(* IEC 61131-3 sources: Elmo_Master/Lasal_PRG/Elmo_EtherCAT_Test_4Axis/Class/GL_9086_1_Slot00, 1 file *)

(* ---- GL_9086_1_Slot00.st ---- *)
//{{ECAT_DEFINES
#define GL_9086_1_SLOT00_ETHERCATSLAVE_PRODUCT_CODE 1196692218
#define GL_9086_1_SLOT00_ETHERCATSLAVE_VENDOR_ID    669
#define GL_9086_1_SLOT00_INPUTS_BYTE0_INDEX		16#6000
#define GL_9086_1_SLOT00_INPUTS_BYTE0_SUBINDEX			1
#define GL_9086_1_SLOT00_INPUTS_BYTE1_INDEX		16#6000
#define GL_9086_1_SLOT00_INPUTS_BYTE1_SUBINDEX			2
#define GL_9086_1_SLOT00_INPUTS_BYTE2_INDEX		16#6000
#define GL_9086_1_SLOT00_INPUTS_BYTE2_SUBINDEX			3
#define GL_9086_1_SLOT00_INPUTS_BYTE3_INDEX		16#6000
#define GL_9086_1_SLOT00_INPUTS_BYTE3_SUBINDEX			4
//}}ECAT_DEFINES

(*!
<Class
	Name               = "GL_9086_1_Slot00"
	Revision           = "0.0"
	RealtimeTask       = "false"
	CyclicTask         = "false"
	BackgroundTask     = "false"
	Sigmatek           = "false"
	OSInterface        = "false"
	HighPriority       = "false"
	Automatic          = "false"
	UpdateMode         = "Prescan"
	SharedCommandTable = "true"
	Objectsize         = "(600,120)"
	Comment            = "GT-12FA">
	<Channels>
		<Server Name="InputS_Byte0" Visualized="false" Initialize="false" WriteProtected="true" Retentive="false" Comment="Input(s)"/>
		<Server Name="InputS_Byte1" Visualized="false" Initialize="false" WriteProtected="true" Retentive="false" Comment="Input(s)"/>
		<Server Name="InputS_Byte2" Visualized="false" Initialize="false" WriteProtected="true" Retentive="false" Comment="Input(s)"/>
		<Server Name="InputS_Byte3" Visualized="false" Initialize="false" WriteProtected="true" Retentive="false" Comment="Input(s)"/>
	</Channels>
	<Network Name="GL_9086_1_Slot00">
		<!-- List of Components in this network -->
		<Components>
			<Object
				Name       = "_base"
				Class      = "ECAT_SlotBase"
				Position   = "(218,120)"
				Visualized = "true"
				Remotely   = "true">
				<Channels>
					<Server Name="ClassState"/>
					<Client Name="ECATSlotIn"/>
					<Client Name="Required" Value="1"/>
					<Client Name="Slot"/>
					<Client Name="SlotIndexInc" Value="0"/>
					<Client Name="ToStdLib"/>
					<Client Name="UseSlotIndexInc" Value="0"/>
				</Channels>
				<AdditionalData>
					<Entry Name="DeviceType" Value="ECAT_SlotBase"/>
					<Entry Name="HWKey" Value="HWD:M_ETHERCAT_MODULE:1:1:0"/>
				</AdditionalData>
			</Object>
		</Components>
		<Comments>
		</Comments>
		<!-- List of Connections in this network -->
		<Connections>
			<Connection Source="this.ClassState" Destination="_base.ClassState" Vertices="(902,210),(730,210),"/>
			<Connection Source="_base.ECATSlotIn" Destination="this.ECATSlotIn" Vertices="(218,210),(38,210),"/>
			<Connection Source="_base.Slot" Destination="this.Slot" Vertices="(218,270),(38,270),"/>
			<Connection Source="_base.SlotIndexInc" Destination="this.SlotIndexInc" Vertices="(218,330),(38,330),"/>
			<Connection Source="_base.UseSlotIndexInc" Destination="this.UseSlotIndexInc" Vertices="(218,390),(38,390),"/>
		</Connections>
		<!-- Headerfiles -->
		<Options>
		</Options>
	</Network>
	<ECAT_SlotModule Type="GT-12FA" ModuleVendor="669" ModuleIdent="1196692218" FileName="..\Runtime\HWConfig\ESI\Crevis EtherCAT IO Module\Crevis_GT-xxxx_V14.xml"/>
	<ECAT_SlotInfoData Type="0" Index="0"/>
</Class>
*)
#pragma using ECAT_SlotBase

GL_9086_1_Slot00 : CLASS
: ECAT_SlotBase
  //Servers:
	InputS_Byte0 	: SvrCh_DINT;
	InputS_Byte1 	: SvrCh_DINT;
	InputS_Byte2 	: SvrCh_DINT;
	InputS_Byte3 	: SvrCh_DINT;
  //Clients:
  //Variables:
  //Functions:
				//! <Function Comment="Overwrite in derived class to set the pdo settings" Name="SetPDOSettings"/>
	FUNCTION VIRTUAL GLOBAL SetPDOSettings
		VAR_OUTPUT
			retcode 	: DINT;
		END_VAR;
  //Tables:
	FUNCTION @STD
		VAR_OUTPUT
			ret_code	: CONFSTATES;
		END_VAR;
	FUNCTION GLOBAL TAB @CT_;
END_CLASS;

FUNCTION VIRTUAL GLOBAL GL_9086_1_Slot00::SetPDOSettings
	VAR_OUTPUT
		retcode 	: DINT;
	END_VAR

	retcode := ECAT_SlotBase::SetPDOSettings();
	if retcode <> 0 then
		return;
	end_if;

	retcode := AddPDOEntry(ECAT_PDO_TYPE_INPUT, #InputS_Byte0.dData, GL_9086_1_SLOT00_INPUTS_BYTE0_INDEX, GL_9086_1_SLOT00_INPUTS_BYTE0_SUBINDEX);
	if retcode <> 0 then
		AddPDOEntryFailed(retcode);
		return;
	end_if;

	retcode := AddPDOEntry(ECAT_PDO_TYPE_INPUT, #InputS_Byte1.dData, GL_9086_1_SLOT00_INPUTS_BYTE1_INDEX, GL_9086_1_SLOT00_INPUTS_BYTE1_SUBINDEX);
	if retcode <> 0 then
		AddPDOEntryFailed(retcode);
		return;
	end_if;

	retcode := AddPDOEntry(ECAT_PDO_TYPE_INPUT, #InputS_Byte2.dData, GL_9086_1_SLOT00_INPUTS_BYTE2_INDEX, GL_9086_1_SLOT00_INPUTS_BYTE2_SUBINDEX);
	if retcode <> 0 then
		AddPDOEntryFailed(retcode);
		return;
	end_if;

	retcode := AddPDOEntry(ECAT_PDO_TYPE_INPUT, #InputS_Byte3.dData, GL_9086_1_SLOT00_INPUTS_BYTE3_INDEX, GL_9086_1_SLOT00_INPUTS_BYTE3_SUBINDEX);
	if retcode <> 0 then
		AddPDOEntryFailed(retcode);
		return;
	end_if;

END_FUNCTION
